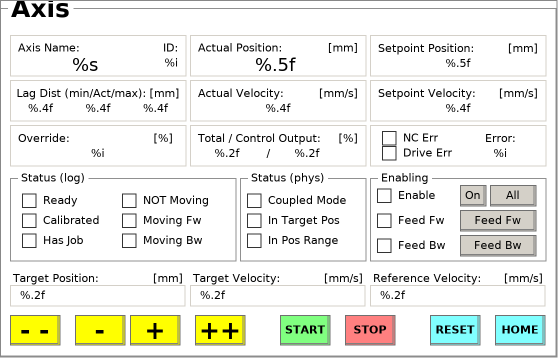
VISUALIZATION PH_NcOnline  // 558x358
VAR_IN_OUT
	stMcAxisOnline			: ST_McAxisOnline;	
END_VAR
VAR
	lrMaxLag				: LREAL;
	lrMinLag                : LREAL;
END_VAR
    Rectangle (2,17 553x339)
    GroupBox (0,0 556x356), "Axis"
        GroupBox (10,170 226x91), "Status (log)"
            Checkbox (10,20 86x21), "Ready", variable: stMcAxisOnline.stStatus.stAxisStatus.Operational
            Checkbox (10,40 86x21), "Calibrated", variable: stMcAxisOnline.stStatus.stAxisStatus.Homed
            Checkbox (10,60 86x21), "Has Job", variable: stMcAxisOnline.stStatus.stAxisStatus.HasJob
            Checkbox (110,20 96x21), "NOT Moving", variable: stMcAxisOnline.stStatus.stAxisStatus.NotMoving
            Checkbox (110,40 96x21), "Moving Fw", variable: stMcAxisOnline.stStatus.stAxisStatus.PositiveDirection
            Checkbox (110,60 96x21), "Moving Bw", variable: stMcAxisOnline.stStatus.stAxisStatus.NegativeDirection
        GroupBox (240,170 126x91), "Status (phys)"
            Checkbox (5,60 116x21), "In Pos Range", variable: stMcAxisOnline.stStatus.stAxisStatus.InPositionArea
            Checkbox (5,40 116x21), "In Target Pos", variable: stMcAxisOnline.stStatus.stAxisStatus.InTargetPosition
            Checkbox (5,20 116x21), "Coupled Mode", variable: stMcAxisOnline.stStatus.stAxisStatus.ProtectedMode
        GroupBox (370,170 176x91), "Enabling"
            Checkbox (5,15 85x21), "Enable", variable: stMcAxisOnline.mcPower.bEnable
            Checkbox (5,40 85x21), "Feed Fw", variable: stMcAxisOnline.mcPower.bEnable_Positive
            Checkbox (5,65 85x21), "Feed Bw", variable: stMcAxisOnline.mcPower.bEnable_Negative
            Button (90,15 26x21), "On"
                toggle stMcAxisOnline.mcPower.bEnable
            Button (90,40 76x21), "Feed Fw"
                toggle stMcAxisOnline.mcPower.bEnable_Positive
            Button (90,65 76x21), "Feed Bw"
                toggle stMcAxisOnline.mcPower.bEnable_Negative
            Button (120,15 46x21), "All"
                OnMouseClick: execute {
                    stMcAxisOnline.mcPower.bEnable				:= TRUE;
                    stMcAxisOnline.mcPower.bEnable_Positive		:= TRUE;
                    stMcAxisOnline.mcPower.bEnable_Negative		:= TRUE;
                    stMcAxisOnline.mcPower.lrOverride			:= 100.0;
                }
        Textfield (370,270 126x17), "Reference Velocity:"
        Textfield (490,270 56x17), "[mm/s]"
        Textfield (370,285 175x21), "%.2f", text variable: stMcAxisOnline.stAxisParameter.fDriveVeloReferenz
            OnMouseClick: write the text variable via Default
        Textfield (10,270 101x17), "Target Position:"
        Textfield (130,270 56x17), "[mm]"
        Textfield (10,285 175x21), "%.2f", text variable: stMcAxisOnline.mcMoveAbsolute.lrPosition
            OnMouseClick: write the text variable via Default
        Textfield (190,270 126x17), "Target Velocity:"
        Textfield (310,270 56x17), "[mm/s]"
        Textfield (190,285 175x21), "%.2f", text variable: stMcAxisOnline.mcMoveAbsolute.lrVelocity
            OnMouseClick: write the text variable via Default
        Group (10,80 176x41)
            Textfield (0,0 176x41)
            Textfield (5,5 166x17), "Lag Dist (min/Act/max): [mm]"
            Textfield (60,20 56x17), "%.4f", text variable: stMcAxisOnline.stStatus.lrPosDiff
            Textfield (120,20 51x17), "%.4f", text variable: stMcAxisOnline.stStatus.lrPosDiff_Max
            Textfield (5,20 51x17), "%.4f", text variable: stMcAxisOnline.stStatus.lrPosDiff_Min
        Group (190,35 176x41)
            Textfield (0,0 176x41)
            Textfield (0,21 171x18), "%.5f", text variable: stMcAxisOnline.stStatus.lrActPos
            Textfield (5,5 91x16), "Actual Position:"
            Textfield (135,5 36x16), "[mm]"
        Textfield (10,35 176x41)
        Textfield (15,56 141x18), "%s", text variable: stMcAxisOnline.stStatus.sAxisName
        Textfield (15,40 91x16), "Axis Name:"
        Group (190,80 176x41)
            Textfield (0,0 176x41)
            Textfield (5,5 91x17), "Actual Velocity:"
            Textfield (5,20 166x17), "%.4f", text variable: stMcAxisOnline.stStatus.lrActVelo
            Textfield (130,5 41x17), "[mm/s]"
        Group (370,80 176x41)
            Textfield (0,0 176x41)
            Textfield (5,5 166x17), "Setpoint Velocity:"
            Textfield (5,20 166x17), "%.4f", text variable: stMcAxisOnline.stStatus.lrSetVelo
            Textfield (130,5 41x17), "[mm/s]"
        Group (370,35 176x41)
            Textfield (0,0 176x41)
            Textfield (5,5 166x17), "Setpoint Position:"
            Textfield (5,20 166x17), "%.5f", text variable: stMcAxisOnline.stStatus.lrSetPos
            Textfield (130,5 41x17), "[mm]"
        Group (10,125 176x41)
            Textfield (0,0 176x41)
            Textfield (5,5 56x17), "Override:"
            Textfield (5,20 166x17), "%i", text variable: stMcAxisOnline.mcPower.lrOverride
                OnMouseClick: write the text variable via Default, min 0, max 100
            Textfield (140,5 26x17), "[%]"
        Group (370,125 176x41)
            Textfield (0,0 176x41), colour toggle: stMcAxisOnline.stStatus.bNcError
            Textfield (90,5 81x17), "Error:"
            Textfield (90,20 81x17), "%i", text variable: stMcAxisOnline.stStatus.udiNcErrorCode
            Checkbox (10,20 71x16), "Drive Err", variable: (stMcAxisOnline.stStatus.udiNcErrorCode AND 16#FF00) = 16#4600
            Checkbox (10,5 66x16), "NC Err", variable: stMcAxisOnline.stStatus.udiNcErrorCode > 0 AND stMcAxisOnline.stStatus.udiNcErrorCode < 18000 AND stMcAxisOnline.stStatus.udiNcErrorCode > 18000
        Button (280,315 50x30), "START"
            tap stMcAxisOnline.mcMoveAbsolute.bExecute
        Button (345,315 50x30), "STOP"
            tap stMcAxisOnline.mcStop.bExecute
        Button (495,315 50x30), "HOME"
            tap stMcAxisOnline.mcHome.bExecute
        Button (430,315 50x30), "RESET"
            tap stMcAxisOnline.mcReset.bExecute
        Button (130,315 50x30), "+"
            tap stMcAxisOnline.mcJog.bSlowForward
        Button (195,315 50x30), "++"
            tap stMcAxisOnline.mcJog.bFastForward
        Button (75,315 50x30), "-"
            tap stMcAxisOnline.mcJog.bSlowBackward
        Button (10,315 50x30), "- -"
            tap stMcAxisOnline.mcJog.bFastBackward
        Textfield (155,40 26x16), "ID:"
        Textfield (155,55 26x16), "%i", text variable: stMcAxisOnline.stStatus.dwAxisId
        Group (190,125 176x41)
            Textfield (0,0 176x41)
            Textfield (5,5 126x17), "Total / Control Output:"
            Textfield (5,20 64x17), "%.2f", text variable: stMcAxisOnline.stStatus.lrTotalOutputInPercent
            Textfield (145,5 26x17), "[%]"
            Textfield (65,20 27x17), "/", text variable: stMcAxisOnline.stStatus.lrTotalOutputInPercent
            Textfield (85,20 64x17), "%.2f", text variable: stMcAxisOnline.stStatus.lrControllerOutputInPercent
END_VISUALIZATION

(* stored: Version 1.1.0.1, ProductVersion 3.1.4026.12
   Visu PH_NcOnline: Id {3c61d9e4-30a3-475e-9c77-b2d9a1d6216d} *)
